RoboDK station: Proyecto_CrisR.rdk

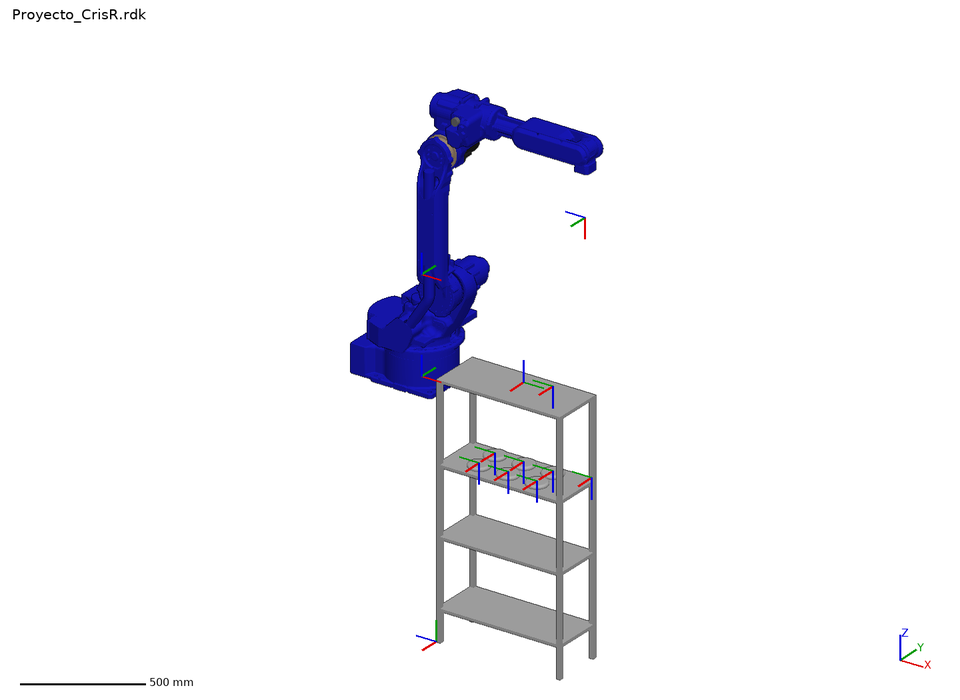
[picture v0: the station drawn from its stored meshes, robots at their saved joint values, targets as dots, program paths as lines]
Station Proyecto_CrisR (saved by RoboDK 5.9.1). Poses are relative to the parent item; angles as X-Y-Z fixed-axis rotations.
  - Python program Prog1 (listed below)
  - frame Frame 1 at (0, 0, 0) mm
    - frame Motoman MH6 Base at (0, 0, 450) mm
      - robot Motoman MH6: 6 axes, payload 6 kg, reach 1422 mm, repeatability 0.08 mm, weight 130 kg
          modified DH rows (alpha deg, a mm, theta deg, d mm): 0, 0, 0, 450; -90, 152, -90, 0; 0, 614, 0, 0; -90, 155, 0, 640; 90, 0, 90, 0; -90, 0, 0, 95
          base shift (0, 0, -450) mm
          joint limits [-170, -90, -175, -180, -45, -360] to [170, 155, 250, 180, 225, 360]; home [0, 0, 0, 0, 0, 0]; saved at [0, 0, 0, 0, 0, 0]
      - frame HOME at (792, 0, 474) mm, rotated rx 0 ry 90 rz 180 deg
  - frame BASE ESTANTERIA at (700, -900, -617) mm, rotated rx 90 ry 0 rz -90 deg
    - object Estanteria at (0, 0, 0) mm, size 250 x 1160 x 600 mm, geometry from Estanteria.stl
    - frame MESA at (-250, 787, -580) mm, rotated rx 90 ry 0 rz 0 deg
      - frame FrameArepa1 at (70, 140, -20) mm
        - object Arepa1 at (0, 0, 0) mm, rotated rx 90 ry 0 rz 0 deg, size 100 x 20 x 99.9 mm, geometry from Arepa.stl
      - frame FrameArepa2 at (180, 140, -20) mm
        - object Arepa2 at (0, 0, 0) mm, rotated rx 90 ry 0 rz 0 deg, size 100 x 20 x 99.9 mm, geometry from Arepa.stl
      - frame FrameArepa3 at (70, 280, -20) mm
        - object Arepa3 at (0, 0, 0) mm, rotated rx 90 ry 0 rz 0 deg, size 100 x 20 x 99.9 mm, geometry from Arepa.stl
      - frame FrameArepa4 at (180, 280, -20) mm
        - object Arepa4 at (0, 0, 0) mm, rotated rx 90 ry 0 rz 0 deg, size 100 x 20 x 99.9 mm, geometry from Arepa.stl
      - frame FrameArepa5 at (70, 420, -20) mm
        - object Arepa5 at (0, 0, 0) mm, rotated rx 90 ry 0 rz 0 deg, size 100 x 20 x 99.9 mm, geometry from Arepa.stl
      - frame FrameArepa6 at (180, 420, -20) mm
        - object Arepa6 at (0, 0, 0) mm, rotated rx 90 ry 0 rz 0 deg, size 100 x 20 x 99.9 mm, geometry from Arepa.stl
      - frame FramePan1 at (70, 140, -392.5) mm
      - frame FramePan2 at (70, 280, -372.5) mm, rotated rx 180 ry 0 rz 0 deg
  - Python program ProgArepa1 (listed below)
  - Python program ProgArepa2 (listed below)
  - Python program ProgArepa3 (listed below)
  - program Prog3 (1 instructions, listed below)

--- Python program Prog1 ---
# Type help("robodk.robolink") or help("robodk.robomath") for more information
# Press F5 to run the script
# Documentation: https://robodk.com/doc/en/RoboDK-API.html
# Reference:     https://robodk.com/doc/en/PythonAPI/robodk.html
# Note: It is not required to keep a copy of this file, your Python script is saved with your RDK project

# You can also use the new version of the API:
from robodk import robolink    # RoboDK API
from robodk import robomath    # Robot toolbox
RDK = robolink.Robolink()

# Forward and backwards compatible use of the RoboDK API:
# Remove these 2 lines to follow python programming guidelines
from robodk import *      # RoboDK API
from robolink import *    # Robot toolbox
# Link to RoboDK
# RDK = Robolink()

# Notify user:
print('To edit this program:\nright click on the Python program, then, select "Edit Python script"')

# Program example:
item = RDK.Item('base')
if item.Valid():
    print('Item selected: ' + item.Name())
    print('Item posistion: ' + repr(item.Pose()))

print('Items in the station:')
itemlist = RDK.ItemList()
print(itemlist)

# Provoking an exception will display the console output if you run this script from RoboDK
raise Exception('Program not edited.')

--- Python program ProgArepa1 ---
from robodk.robolink import *    # API para comunicarte con RoboDK
from robodk.robomath import *    # Funciones matemáticas
import math

#------------------------------------------------
# 1) Conexión a RoboDK e inicialización
#------------------------------------------------

RDK = Robolink()

# Elegir un robot (si hay varios, aparece un popup)
robot = RDK.ItemUserPick("Selecciona un robot", ITEM_TYPE_ROBOT)
#if not robot.Valid():
#    raise Exception("No se ha seleccionado un robot válido.")

# Conectar al robot físico
#if not robot.Connect():
#    raise Exception("No se pudo conectar al robot. Verifica que esté en modo remoto y que la configuración sea correcta.")

# Confirmar conexión
#if not robot.ConnectedState():
#    ("El robot no está conectado correctamente. Revisa la conexión.")

print("Robot conectado correctamente.")

#gripper_name = "Gripper v7"  # Cambia por el nombre de tu gripper
#gripper = RDK.Item(gripper_name, ITEM_TYPE_TOOL)
#if not gripper.Valid():
#    raise Exception(f'No se encontró el gripper "{gripper_name}" en la estación.')

# Establecer el gripper como la herramienta activa
#robot.setTool(gripper)

#------------------------------------------------
# 2) Cargar el Frame
#------------------------------------------------
frame_name2 = "HOME"
frame2 = RDK.Item(frame_name2, ITEM_TYPE_FRAME)
if not frame2.Valid():
    raise Exception(f'No se encontró el Frame "{frame_name2}" en la estación.')

robot.setPoseFrame(frame2)
robot.setPoseTool(robot.PoseTool())

# Ajustes de velocidad y blending
robot.setSpeed(300)   # mm/s
robot.setRounding(5)  # mm

robot.MoveL(transl(0, 0, 0))

#frame_Arepa1 = "FrameArepa1"
#frameArepa1 = RDK.Item(frame_Arepa1, ITEM_TYPE_FRAME)
#if not frameArepa1.Valid():
#    raise Exception(f'No se encontró el Frame "{frame_Arepa1}" en la estación.')


#arepa = RDK.Item("Arepa1", ITEM_TYPE_OBJECT)  # El nombre del objeto STL debe ser correcto
#if not arepa.Valid():
#    raise Exception(f'No se encontró el objeto "Arepa1" en la estación.')

frame_name = "MESA"
frame = RDK.Item(frame_name, ITEM_TYPE_FRAME)
if not frame.Valid():
    raise Exception(f'No se encontró el Frame "{frame_name}" en la estación.')

robot.setPoseFrame(frame)
robot.setPoseTool(robot.PoseTool())

# Ajustes de velocidad y blending
robot.setSpeed(300)   # mm/s
robot.setRounding(5)  # mm

#------------------------------------------------
#               MOVIMIENTO DE AREPA
#------------------------------------------------

robot.MoveL(transl(-100, 0, -50))
robot.MoveL(transl(-100, 140, -50))
robot.MoveL(transl(70, 140, -50))
robot.MoveL(transl(70, 140, 0))
#arepa.setParent(gripper)
robot.MoveL(transl(70, 140, -50))
robot.MoveL(transl(-100, 140, -50))

frame_Pan1 = "FramePan1"
framePan1 = RDK.Item(frame_Pan1, ITEM_TYPE_FRAME)
if not framePan1.Valid():
    raise Exception(f'No se encontró el Frame "{frame_Pan1}" en la estación.')

robot.setPoseFrame(framePan1)
robot.setPoseTool(robot.PoseTool())

# Ajustes de velocidad y blending
robot.setSpeed(300)   # mm/s
robot.setRounding(5)  # mm

robot.MoveL(transl(-270, 0, -50))
robot.MoveL(transl(0, 0, -50))
robot.MoveL(transl(0, 0, 0))
#arepa.setParent(framePan1)
robot.MoveL(transl(0, 0, -50))
robot.MoveL(transl(-270, 0, -50))

frame_name2 = "HOME"
frame2 = RDK.Item(frame_name2, ITEM_TYPE_FRAME)
if not frame2.Valid():
    raise Exception(f'No se encontró el Frame "{frame_name2}" en la estación.')

robot.setPoseFrame(frame2)
robot.setPoseTool(robot.PoseTool())

# Ajustes de velocidad y blending
robot.setSpeed(300)   # mm/s
robot.setRounding(5)  # mm

robot.MoveJ(transl(0, 0, 0))

frame_Pan1 = "FramePan1"
framePan1 = RDK.Item(frame_Pan1, ITEM_TYPE_FRAME)
if not framePan1.Valid():
    raise Exception(f'No se encontró el Frame "{frame_Pan1}" en la estación.')

robot.setPoseFrame(framePan1)
robot.setPoseTool(robot.PoseTool())

# Ajustes de velocidad y blending
robot.setSpeed(300)   # mm/s
robot.setRounding(5)  # mm

robot.MoveL(transl(-270, 0, -50))
robot.MoveL(transl(0, 0, -50))
robot.MoveL(transl(0, 0, 0))
#arepa.setParent(gripper)
robot.MoveL(transl(0, 0, -200))
#joints_actuales = robot.Joints().list()
#joints_actuales[5] += 180
#robot.MoveJ(joints_actuales)

frame_Pan2 = "FramePan2"
framePan2 = RDK.Item(frame_Pan2, ITEM_TYPE_FRAME)
if not framePan2.Valid():
    raise Exception(f'No se encontró el Frame "{frame_Pan2}" en la estación.')

robot.setPoseFrame(framePan2)
robot.setPoseTool(robot.PoseTool())

# Ajustes de velocidad y blending
robot.setSpeed(300)   # mm/s
robot.setRounding(5)  # mm

#robot.MoveL(transl(0, 0, 200))
#robot.MoveL(transl(0, 0, 0))
#arepa.setParent(framePan2)
#robot.MoveL(transl(0, 0, 200))


#------------------------------------------------
#                VUELTA A HOME
#------------------------------------------------

frame_name2 = "HOME"
frame2 = RDK.Item(frame_name2, ITEM_TYPE_FRAME)
if not frame2.Valid():
    raise Exception(f'No se encontró el Frame "{frame_name2}" en la estación.')

robot.setPoseFrame(frame2)
robot.setPoseTool(robot.PoseTool())

# Ajustes de velocidad y blending
robot.setSpeed(300)   # mm/s
robot.setRounding(5)  # mm

robot.MoveJ(transl(0, 0, 0))

#arepa.setParent(frameArepa1)

--- Python program ProgArepa2 ---
from robodk.robolink import *    # API para comunicarte con RoboDK
from robodk.robomath import *    # Funciones matemáticas
import math

#------------------------------------------------
# 1) Conexión a RoboDK e inicialización
#------------------------------------------------

RDK = Robolink()

# Elegir un robot (si hay varios, aparece un popup)
robot = RDK.ItemUserPick("Selecciona un robot", ITEM_TYPE_ROBOT)
#if not robot.Valid():
 #   raise Exception("No se ha seleccionado un robot válido.")

# Conectar al robot físico
#if not robot.Connect():
#    raise Exception("No se pudo conectar al robot. Verifica que esté en modo remoto y que la configuración sea correcta.")

# Confirmar conexión
#if not robot.ConnectedState():
 #   ("El robot no está conectado correctamente. Revisa la conexión.")

print("Robot conectado correctamente.")

gripper_name = "Gripper v7"  # Cambia por el nombre de tu gripper
gripper = RDK.Item(gripper_name, ITEM_TYPE_TOOL)
if not gripper.Valid():
    raise Exception(f'No se encontró el gripper "{gripper_name}" en la estación.')

# Establecer el gripper como la herramienta activa
robot.setTool(gripper)

#------------------------------------------------
# 2) Cargar el Frame
#------------------------------------------------
frame_name2 = "HOME"
frame2 = RDK.Item(frame_name2, ITEM_TYPE_FRAME)
if not frame2.Valid():
    raise Exception(f'No se encontró el Frame "{frame_name2}" en la estación.')

frame_Arepa1 = "FrameArepa2"
frameArepa1 = RDK.Item(frame_Arepa1, ITEM_TYPE_FRAME)
if not frameArepa1.Valid():
    raise Exception(f'No se encontró el Frame "{frame_Arepa1}" en la estación.')

frame_Pan1 = "FramePan1"
framePan1 = RDK.Item(frame_Pan1, ITEM_TYPE_FRAME)
if not framePan1.Valid():
    raise Exception(f'No se encontró el Frame "{frame_Pan1}" en la estación.')

frame_Pan2 = "FramePan2"
framePan2 = RDK.Item(frame_Pan2, ITEM_TYPE_FRAME)
if not framePan2.Valid():
    raise Exception(f'No se encontró el Frame "{frame_Pan2}" en la estación.')


arepa = RDK.Item("Arepa2", ITEM_TYPE_OBJECT)  # El nombre del objeto STL debe ser correcto
if not arepa.Valid():
    raise Exception(f'No se encontró el objeto "Arepa1" en la estación.')

robot.setPoseFrame(frame2)
robot.setPoseTool(robot.PoseTool())
joints_actuales = robot.Joints().list()

# Ajustes de velocidad y blending
robot.setSpeed(300)   # mm/s
robot.setRounding(5)  # mm

robot.MoveL(transl(0, 0, 0))


frame_name = "MESA"
frame = RDK.Item(frame_name, ITEM_TYPE_FRAME)
if not frame.Valid():
    raise Exception(f'No se encontró el Frame "{frame_name}" en la estación.')

robot.setPoseFrame(frame)
robot.setPoseTool(robot.PoseTool())

# Ajustes de velocidad y blending
robot.setSpeed(300)   # mm/s
robot.setRounding(5)  # mm

#------------------------------------------------
# 3) Parámetros del cuarto de círculo
#------------------------------------------------
num_points = 180
radius = 150
z_surface = 0
z_safe = -50

robot.MoveL(transl(-100, 0, -50))
robot.MoveL(transl(-100, 140, -50))
robot.MoveL(transl(180, 140, -50))
robot.MoveL(transl(180, 140, 0))
arepa.setParent(gripper)
robot.MoveL(transl(180, 140, -50))
robot.MoveL(transl(-100, 140, -50))

robot.setPoseFrame(framePan1)
robot.MoveL(transl(-270, 0, -50))
robot.MoveL(transl(0, 0, -50))
robot.MoveL(transl(0, 0, 0))
arepa.setParent(framePan1)
robot.MoveL(transl(0, 0, -50))
robot.MoveL(transl(-270, 0, -50))

robot.setPoseFrame(frame2)
robot.MoveJ(transl(0, 0, 0))

robot.setPoseFrame(framePan1)
robot.MoveL(transl(-270, 0, -50))
robot.MoveL(transl(0, 0, -50))
robot.MoveL(transl(0, 0, 0))
arepa.setParent(gripper)
robot.MoveL(transl(0, 0, -200))
joints_actuales = robot.Joints().list()
joints_actuales[5] += 180
robot.MoveJ(joints_actuales)

robot.setPoseFrame(framePan2)
robot.MoveL(transl(0, 0, 200))
robot.MoveL(transl(0, 0, 0))
arepa.setParent(framePan2)
robot.MoveL(transl(0, 0, 50))

#------------------------------------------------
#                VUELTA A HOME
#------------------------------------------------

robot.setPoseFrame(frame2)
robot.MoveJ(transl(0, 0, 0))

arepa.setParent(frameArepa1)

--- Python program ProgArepa3 ---
from robodk.robolink import *    # API para comunicarte con RoboDK
from robodk.robomath import *    # Funciones matemáticas
import math

#------------------------------------------------
# 1) Conexión a RoboDK e inicialización
#------------------------------------------------

RDK = Robolink()

# Elegir un robot (si hay varios, aparece un popup)
robot = RDK.ItemUserPick("Selecciona un robot", ITEM_TYPE_ROBOT)
#if not robot.Valid():
 #   raise Exception("No se ha seleccionado un robot válido.")

# Conectar al robot físico
#if not robot.Connect():
#    raise Exception("No se pudo conectar al robot. Verifica que esté en modo remoto y que la configuración sea correcta.")

# Confirmar conexión
#if not robot.ConnectedState():
 #   ("El robot no está conectado correctamente. Revisa la conexión.")

print("Robot conectado correctamente.")

gripper_name = "Gripper v7"  # Cambia por el nombre de tu gripper
gripper = RDK.Item(gripper_name, ITEM_TYPE_TOOL)
if not gripper.Valid():
    raise Exception(f'No se encontró el gripper "{gripper_name}" en la estación.')

# Establecer el gripper como la herramienta activa
robot.setTool(gripper)

#------------------------------------------------
# 2) Cargar el Frame
#------------------------------------------------
frame_name2 = "HOME"
frame2 = RDK.Item(frame_name2, ITEM_TYPE_FRAME)
if not frame2.Valid():
    raise Exception(f'No se encontró el Frame "{frame_name2}" en la estación.')

frame_Arepa1 = "FrameArepa3"
frameArepa1 = RDK.Item(frame_Arepa1, ITEM_TYPE_FRAME)
if not frameArepa1.Valid():
    raise Exception(f'No se encontró el Frame "{frame_Arepa1}" en la estación.')

frame_Pan1 = "FramePan1"
framePan1 = RDK.Item(frame_Pan1, ITEM_TYPE_FRAME)
if not framePan1.Valid():
    raise Exception(f'No se encontró el Frame "{frame_Pan1}" en la estación.')

frame_Pan2 = "FramePan2"
framePan2 = RDK.Item(frame_Pan2, ITEM_TYPE_FRAME)
if not framePan2.Valid():
    raise Exception(f'No se encontró el Frame "{frame_Pan2}" en la estación.')


arepa = RDK.Item("Arepa3", ITEM_TYPE_OBJECT)  # El nombre del objeto STL debe ser correcto
if not arepa.Valid():
    raise Exception(f'No se encontró el objeto "Arepa1" en la estación.')

robot.setPoseFrame(frame2)
robot.setPoseTool(robot.PoseTool())
joints_actuales = robot.Joints().list()

# Ajustes de velocidad y blending
robot.setSpeed(300)   # mm/s
robot.setRounding(5)  # mm

robot.MoveL(transl(0, 0, 0))


frame_name = "MESA"
frame = RDK.Item(frame_name, ITEM_TYPE_FRAME)
if not frame.Valid():
    raise Exception(f'No se encontró el Frame "{frame_name}" en la estación.')

robot.setPoseFrame(frame)
robot.setPoseTool(robot.PoseTool())

# Ajustes de velocidad y blending
robot.setSpeed(300)   # mm/s
robot.setRounding(5)  # mm

#------------------------------------------------
# 3) Parámetros del cuarto de círculo
#------------------------------------------------

robot.MoveL(transl(-100, 0, -50))
robot.MoveL(transl(-100, 280, -50))
robot.MoveL(transl(70, 280, -50))
robot.MoveL(transl(70, 280, 0))
arepa.setParent(gripper)
robot.MoveL(transl(70, 280, -50))
robot.MoveL(transl(-100, 280, -50))

robot.setPoseFrame(framePan1)
robot.MoveL(transl(-270, 0, -50))
robot.MoveL(transl(0, 0, -50))
robot.MoveL(transl(0, 0, 0))
arepa.setParent(framePan1)
robot.MoveL(transl(0, 0, -50))
robot.MoveL(transl(-270, 0, -50))

robot.setPoseFrame(frame2)
robot.setPoseTool(robot.PoseTool())
robot.MoveJ(transl(0, 0, 0))

robot.setPoseFrame(framePan1)
robot.MoveL(transl(-270, 0, -50))
robot.MoveL(transl(0, 0, -50))
robot.MoveL(transl(0, 0, 0))
arepa.setParent(gripper)
robot.MoveL(transl(0, 0, -200))
joints_actuales = robot.Joints().list()
joints_actuales[5] += 180
robot.MoveJ(joints_actuales)

robot.setPoseFrame(framePan2)
robot.MoveL(transl(0, 0, 200))
robot.MoveL(transl(0, 0, 0))
arepa.setParent(framePan2)
robot.MoveL(transl(0, 0, 50))

#------------------------------------------------
#                VUELTA A HOME
#------------------------------------------------

robot.setPoseFrame(frame2)
robot.MoveJ(transl(0, 0, 0))

arepa.setParent(frameArepa1)

--- program Prog3 (robot Motoman MH6) ---
  Wait DI1=0
